TYPE ST115_Feeder_e : ST110_Feeder_e;
END_TYPE

(* stored: Version 1.1.0.1, ProductVersion 3.1.4024.6
   DUT ST115_Feeder_e: Id {cc37ee37-bc3e-4846-8d73-2e341d83d408} *)
